    PROC main()
        Path_Draw;
    ENDPROC
    LOCAL PROC Path_Draw()
        MoveL point_0_clearance,v1000,fine,MyTool\WObj:=Workobject_1;
        MoveL point_0_contact,v1000,fine,MyTool\WObj:=Workobject_1;
        MoveL point_1_contact,v1000,fine,MyTool\WObj:=Workobject_1;
        MoveL point_1_clearance,v1000,fine,MyTool\WObj:=Workobject_1;
        MoveL point_2_clearance,v1000,fine,MyTool\WObj:=Workobject_1;
        MoveL point_2_contact,v1000,fine,MyTool\WObj:=Workobject_1;
        MoveL point_3_contact,v1000,fine,MyTool\WObj:=Workobject_1;
        MoveL point_3_clearance,v1000,fine,MyTool\WObj:=Workobject_1;
        MoveL point_4_clearance,v1000,fine,MyTool\WObj:=Workobject_1;
        MoveL point_4_contact,v1000,fine,MyTool\WObj:=Workobject_1;
        MoveL point_5_contact,v1000,fine,MyTool\WObj:=Workobject_1;
        MoveL point_5_clearance,v1000,fine,MyTool\WObj:=Workobject_1;
        MoveL point_6_clearance,v1000,fine,MyTool\WObj:=Workobject_1;
        MoveL point_6_contact,v1000,fine,MyTool\WObj:=Workobject_1;
        MoveL point_7_contact,v1000,fine,MyTool\WObj:=Workobject_1;
        MoveL point_7_clearance,v1000,fine,MyTool\WObj:=Workobject_1;
        MoveL point_8_clearance,v1000,fine,MyTool\WObj:=Workobject_1;
        MoveL point_8_contact,v1000,fine,MyTool\WObj:=Workobject_1;
        MoveL point_9_contact,v1000,fine,MyTool\WObj:=Workobject_1;
        MoveL point_9_clearance,v1000,fine,MyTool\WObj:=Workobject_1;
        MoveL point_10_clearance,v1000,fine,MyTool\WObj:=Workobject_1;
        MoveL point_10_contact,v1000,fine,MyTool\WObj:=Workobject_1;
        MoveL point_11_contact,v1000,fine,MyTool\WObj:=Workobject_1;
        MoveL point_11_clearance,v1000,fine,MyTool\WObj:=Workobject_1;
        MoveL point_12_clearance,v1000,fine,MyTool\WObj:=Workobject_1;
        MoveL point_12_contact,v1000,fine,MyTool\WObj:=Workobject_1;
        MoveL point_13_contact,v1000,fine,MyTool\WObj:=Workobject_1;
        MoveL point_13_clearance,v1000,fine,MyTool\WObj:=Workobject_1;
        MoveL point_14_clearance,v1000,fine,MyTool\WObj:=Workobject_1;
        MoveL point_14_contact,v1000,fine,MyTool\WObj:=Workobject_1;
        MoveL point_15_contact,v1000,fine,MyTool\WObj:=Workobject_1;
        MoveL point_15_clearance,v1000,fine,MyTool\WObj:=Workobject_1;
        MoveL point_16_clearance,v1000,fine,MyTool\WObj:=Workobject_1;
        MoveL point_16_contact,v1000,fine,MyTool\WObj:=Workobject_1;
        MoveL point_17_contact,v1000,fine,MyTool\WObj:=Workobject_1;
        MoveL point_17_clearance,v1000,fine,MyTool\WObj:=Workobject_1;
        MoveL point_18_clearance,v1000,fine,MyTool\WObj:=Workobject_1;
        MoveL point_18_contact,v1000,fine,MyTool\WObj:=Workobject_1;
        MoveL point_19_contact,v1000,fine,MyTool\WObj:=Workobject_1;
        MoveL point_19_clearance,v1000,fine,MyTool\WObj:=Workobject_1;
        MoveL point_20_clearance,v1000,fine,MyTool\WObj:=Workobject_1;
        MoveL point_20_contact,v1000,fine,MyTool\WObj:=Workobject_1;
        MoveL point_21_contact,v1000,fine,MyTool\WObj:=Workobject_1;
        MoveL point_21_clearance,v1000,fine,MyTool\WObj:=Workobject_1;
        MoveL point_22_clearance,v1000,fine,MyTool\WObj:=Workobject_1;
        MoveL point_22_contact,v1000,fine,MyTool\WObj:=Workobject_1;
        MoveL point_23_contact,v1000,fine,MyTool\WObj:=Workobject_1;
        MoveL point_23_clearance,v1000,fine,MyTool\WObj:=Workobject_1;
        MoveL point_24_clearance,v1000,fine,MyTool\WObj:=Workobject_1;
        MoveL point_24_contact,v1000,fine,MyTool\WObj:=Workobject_1;
        MoveL point_25_contact,v1000,fine,MyTool\WObj:=Workobject_1;
        MoveL point_25_clearance,v1000,fine,MyTool\WObj:=Workobject_1;
        MoveL point_26_clearance,v1000,fine,MyTool\WObj:=Workobject_1;
        MoveL point_26_contact,v1000,fine,MyTool\WObj:=Workobject_1;
        MoveL point_27_contact,v1000,fine,MyTool\WObj:=Workobject_1;
        MoveL point_27_clearance,v1000,fine,MyTool\WObj:=Workobject_1;
        MoveL point_28_clearance,v1000,fine,MyTool\WObj:=Workobject_1;
        MoveL point_28_contact,v1000,fine,MyTool\WObj:=Workobject_1;
        MoveL point_29_contact,v1000,fine,MyTool\WObj:=Workobject_1;
        MoveL point_29_clearance,v1000,fine,MyTool\WObj:=Workobject_1;
        MoveL point_30_clearance,v1000,fine,MyTool\WObj:=Workobject_1;
        MoveL point_30_contact,v1000,fine,MyTool\WObj:=Workobject_1;
        MoveL point_31_contact,v1000,fine,MyTool\WObj:=Workobject_1;
        MoveL point_31_clearance,v1000,fine,MyTool\WObj:=Workobject_1;
        MoveL point_32_clearance,v1000,fine,MyTool\WObj:=Workobject_1;
        MoveL point_32_contact,v1000,fine,MyTool\WObj:=Workobject_1;
        MoveL point_33_contact,v1000,fine,MyTool\WObj:=Workobject_1;
        MoveL point_33_clearance,v1000,fine,MyTool\WObj:=Workobject_1;
        MoveL point_34_clearance,v1000,fine,MyTool\WObj:=Workobject_1;
        MoveL point_34_contact,v1000,fine,MyTool\WObj:=Workobject_1;
        MoveL point_35_contact,v1000,fine,MyTool\WObj:=Workobject_1;
        MoveL point_35_clearance,v1000,fine,MyTool\WObj:=Workobject_1;
        MoveL point_36_clearance,v1000,fine,MyTool\WObj:=Workobject_1;
        MoveL point_36_contact,v1000,fine,MyTool\WObj:=Workobject_1;
        MoveL point_37_contact,v1000,fine,MyTool\WObj:=Workobject_1;
        MoveL point_37_clearance,v1000,fine,MyTool\WObj:=Workobject_1;
        MoveL point_38_clearance,v1000,fine,MyTool\WObj:=Workobject_1;
        MoveL point_38_contact,v1000,fine,MyTool\WObj:=Workobject_1;
        MoveL point_39_contact,v1000,fine,MyTool\WObj:=Workobject_1;
        MoveL point_39_clearance,v1000,fine,MyTool\WObj:=Workobject_1;
        MoveL point_40_clearance,v1000,fine,MyTool\WObj:=Workobject_1;
        MoveL point_40_contact,v1000,fine,MyTool\WObj:=Workobject_1;
        MoveL point_41_contact,v1000,fine,MyTool\WObj:=Workobject_1;
        MoveL point_41_clearance,v1000,fine,MyTool\WObj:=Workobject_1;
        MoveL point_42_clearance,v1000,fine,MyTool\WObj:=Workobject_1;
        MoveL point_42_contact,v1000,fine,MyTool\WObj:=Workobject_1;
        MoveL point_43_contact,v1000,fine,MyTool\WObj:=Workobject_1;
        MoveL point_43_clearance,v1000,fine,MyTool\WObj:=Workobject_1;
        MoveL point_44_clearance,v1000,fine,MyTool\WObj:=Workobject_1;
        MoveL point_44_contact,v1000,fine,MyTool\WObj:=Workobject_1;
        MoveL point_45_contact,v1000,fine,MyTool\WObj:=Workobject_1;
        MoveL point_45_clearance,v1000,fine,MyTool\WObj:=Workobject_1;
        MoveL point_46_clearance,v1000,fine,MyTool\WObj:=Workobject_1;
        MoveL point_46_contact,v1000,fine,MyTool\WObj:=Workobject_1;
        MoveL point_47_contact,v1000,fine,MyTool\WObj:=Workobject_1;
        MoveL point_47_clearance,v1000,fine,MyTool\WObj:=Workobject_1;
        MoveL point_48_clearance,v1000,fine,MyTool\WObj:=Workobject_1;
        MoveL point_48_contact,v1000,fine,MyTool\WObj:=Workobject_1;
        MoveL point_49_contact,v1000,fine,MyTool\WObj:=Workobject_1;
        MoveL point_49_clearance,v1000,fine,MyTool\WObj:=Workobject_1;
        MoveL point_50_clearance,v1000,fine,MyTool\WObj:=Workobject_1;
        MoveL point_50_contact,v1000,fine,MyTool\WObj:=Workobject_1;
        MoveL point_51_contact,v1000,fine,MyTool\WObj:=Workobject_1;
        MoveL point_51_clearance,v1000,fine,MyTool\WObj:=Workobject_1;
        MoveL point_52_clearance,v1000,fine,MyTool\WObj:=Workobject_1;
        MoveL point_52_contact,v1000,fine,MyTool\WObj:=Workobject_1;
        MoveL point_53_contact,v1000,fine,MyTool\WObj:=Workobject_1;
        MoveL point_53_clearance,v1000,fine,MyTool\WObj:=Workobject_1;
        MoveL point_54_clearance,v1000,fine,MyTool\WObj:=Workobject_1;
        MoveL point_54_contact,v1000,fine,MyTool\WObj:=Workobject_1;
        MoveL point_55_contact,v1000,fine,MyTool\WObj:=Workobject_1;
        MoveL point_55_clearance,v1000,fine,MyTool\WObj:=Workobject_1;
        MoveL point_56_clearance,v1000,fine,MyTool\WObj:=Workobject_1;
        MoveL point_56_contact,v1000,fine,MyTool\WObj:=Workobject_1;
        MoveL point_57_contact,v1000,fine,MyTool\WObj:=Workobject_1;
        MoveL point_57_clearance,v1000,fine,MyTool\WObj:=Workobject_1;
        MoveL point_58_clearance,v1000,fine,MyTool\WObj:=Workobject_1;
        MoveL point_58_contact,v1000,fine,MyTool\WObj:=Workobject_1;
        MoveL point_59_contact,v1000,fine,MyTool\WObj:=Workobject_1;
        MoveL point_59_clearance,v1000,fine,MyTool\WObj:=Workobject_1;
        MoveL point_60_clearance,v1000,fine,MyTool\WObj:=Workobject_1;
        MoveL point_60_contact,v1000,fine,MyTool\WObj:=Workobject_1;
        MoveL point_61_contact,v1000,fine,MyTool\WObj:=Workobject_1;
        MoveL point_61_clearance,v1000,fine,MyTool\WObj:=Workobject_1;
        MoveL point_62_clearance,v1000,fine,MyTool\WObj:=Workobject_1;
        MoveL point_62_contact,v1000,fine,MyTool\WObj:=Workobject_1;
        MoveL point_63_contact,v1000,fine,MyTool\WObj:=Workobject_1;
        MoveL point_63_clearance,v1000,fine,MyTool\WObj:=Workobject_1;
        MoveL point_64_clearance,v1000,fine,MyTool\WObj:=Workobject_1;
        MoveL point_64_contact,v1000,fine,MyTool\WObj:=Workobject_1;
        MoveL point_65_contact,v1000,fine,MyTool\WObj:=Workobject_1;
        MoveL point_65_clearance,v1000,fine,MyTool\WObj:=Workobject_1;
        MoveL point_66_clearance,v1000,fine,MyTool\WObj:=Workobject_1;
        MoveL point_66_contact,v1000,fine,MyTool\WObj:=Workobject_1;
        MoveL point_67_contact,v1000,fine,MyTool\WObj:=Workobject_1;
        MoveL point_67_clearance,v1000,fine,MyTool\WObj:=Workobject_1;
        MoveL point_68_clearance,v1000,fine,MyTool\WObj:=Workobject_1;
        MoveL point_68_contact,v1000,fine,MyTool\WObj:=Workobject_1;
        MoveL point_69_contact,v1000,fine,MyTool\WObj:=Workobject_1;
        MoveL point_69_clearance,v1000,fine,MyTool\WObj:=Workobject_1;
        MoveL point_70_clearance,v1000,fine,MyTool\WObj:=Workobject_1;
        MoveL point_70_contact,v1000,fine,MyTool\WObj:=Workobject_1;
        MoveL point_71_contact,v1000,fine,MyTool\WObj:=Workobject_1;
        MoveL point_71_clearance,v1000,fine,MyTool\WObj:=Workobject_1;
        MoveL point_72_clearance,v1000,fine,MyTool\WObj:=Workobject_1;
        MoveL point_72_contact,v1000,fine,MyTool\WObj:=Workobject_1;
        MoveL point_73_contact,v1000,fine,MyTool\WObj:=Workobject_1;
        MoveL point_73_clearance,v1000,fine,MyTool\WObj:=Workobject_1;
        MoveL point_74_clearance,v1000,fine,MyTool\WObj:=Workobject_1;
        MoveL point_74_contact,v1000,fine,MyTool\WObj:=Workobject_1;
        MoveL point_75_contact,v1000,fine,MyTool\WObj:=Workobject_1;
        MoveL point_75_clearance,v1000,fine,MyTool\WObj:=Workobject_1;
        MoveL point_76_clearance,v1000,fine,MyTool\WObj:=Workobject_1;
        MoveL point_76_contact,v1000,fine,MyTool\WObj:=Workobject_1;
        MoveL point_77_contact,v1000,fine,MyTool\WObj:=Workobject_1;
        MoveL point_77_clearance,v1000,fine,MyTool\WObj:=Workobject_1;
        MoveL point_78_clearance,v1000,fine,MyTool\WObj:=Workobject_1;
        MoveL point_78_contact,v1000,fine,MyTool\WObj:=Workobject_1;
        MoveL point_79_contact,v1000,fine,MyTool\WObj:=Workobject_1;
        MoveL point_79_clearance,v1000,fine,MyTool\WObj:=Workobject_1;
        MoveL point_80_clearance,v1000,fine,MyTool\WObj:=Workobject_1;
        MoveL point_80_contact,v1000,fine,MyTool\WObj:=Workobject_1;
        MoveL point_81_contact,v1000,fine,MyTool\WObj:=Workobject_1;
        MoveL point_81_clearance,v1000,fine,MyTool\WObj:=Workobject_1;
        MoveL point_82_clearance,v1000,fine,MyTool\WObj:=Workobject_1;
        MoveL point_82_contact,v1000,fine,MyTool\WObj:=Workobject_1;
        MoveL point_83_contact,v1000,fine,MyTool\WObj:=Workobject_1;
        MoveL point_83_clearance,v1000,fine,MyTool\WObj:=Workobject_1;
        MoveL point_84_clearance,v1000,fine,MyTool\WObj:=Workobject_1;
        MoveL point_84_contact,v1000,fine,MyTool\WObj:=Workobject_1;
        MoveL point_85_contact,v1000,fine,MyTool\WObj:=Workobject_1;
        MoveL point_85_clearance,v1000,fine,MyTool\WObj:=Workobject_1;
        MoveL point_86_clearance,v1000,fine,MyTool\WObj:=Workobject_1;
        MoveL point_86_contact,v1000,fine,MyTool\WObj:=Workobject_1;
        MoveL point_87_contact,v1000,fine,MyTool\WObj:=Workobject_1;
        MoveL point_87_clearance,v1000,fine,MyTool\WObj:=Workobject_1;
        MoveL point_88_clearance,v1000,fine,MyTool\WObj:=Workobject_1;
        MoveL point_88_contact,v1000,fine,MyTool\WObj:=Workobject_1;
        MoveL point_89_contact,v1000,fine,MyTool\WObj:=Workobject_1;
        MoveL point_89_clearance,v1000,fine,MyTool\WObj:=Workobject_1;
        MoveL point_90_clearance,v1000,fine,MyTool\WObj:=Workobject_1;
        MoveL point_90_contact,v1000,fine,MyTool\WObj:=Workobject_1;
        MoveL point_91_contact,v1000,fine,MyTool\WObj:=Workobject_1;
        MoveL point_91_clearance,v1000,fine,MyTool\WObj:=Workobject_1;
        MoveL point_92_clearance,v1000,fine,MyTool\WObj:=Workobject_1;
        MoveL point_92_contact,v1000,fine,MyTool\WObj:=Workobject_1;
        MoveL point_93_contact,v1000,fine,MyTool\WObj:=Workobject_1;
        MoveL point_93_clearance,v1000,fine,MyTool\WObj:=Workobject_1;
        MoveL point_94_clearance,v1000,fine,MyTool\WObj:=Workobject_1;
        MoveL point_94_contact,v1000,fine,MyTool\WObj:=Workobject_1;
        MoveL point_95_contact,v1000,fine,MyTool\WObj:=Workobject_1;
        MoveL point_95_clearance,v1000,fine,MyTool\WObj:=Workobject_1;
        MoveL point_96_clearance,v1000,fine,MyTool\WObj:=Workobject_1;
        MoveL point_96_contact,v1000,fine,MyTool\WObj:=Workobject_1;
        MoveL point_97_contact,v1000,fine,MyTool\WObj:=Workobject_1;
        MoveL point_97_clearance,v1000,fine,MyTool\WObj:=Workobject_1;
        MoveL point_98_clearance,v1000,fine,MyTool\WObj:=Workobject_1;
        MoveL point_98_contact,v1000,fine,MyTool\WObj:=Workobject_1;
        MoveL point_99_contact,v1000,fine,MyTool\WObj:=Workobject_1;
        MoveL point_99_clearance,v1000,fine,MyTool\WObj:=Workobject_1;
        MoveL point_100_clearance,v1000,fine,MyTool\WObj:=Workobject_1;
        MoveL point_100_contact,v1000,fine,MyTool\WObj:=Workobject_1;
        MoveL point_101_contact,v1000,fine,MyTool\WObj:=Workobject_1;
        MoveL point_101_clearance,v1000,fine,MyTool\WObj:=Workobject_1;
        MoveL point_102_clearance,v1000,fine,MyTool\WObj:=Workobject_1;
        MoveL point_102_contact,v1000,fine,MyTool\WObj:=Workobject_1;
        MoveL point_103_contact,v1000,fine,MyTool\WObj:=Workobject_1;
        MoveL point_103_clearance,v1000,fine,MyTool\WObj:=Workobject_1;
        MoveL point_104_clearance,v1000,fine,MyTool\WObj:=Workobject_1;
        MoveL point_104_contact,v1000,fine,MyTool\WObj:=Workobject_1;
        MoveL point_105_contact,v1000,fine,MyTool\WObj:=Workobject_1;
        MoveL point_105_clearance,v1000,fine,MyTool\WObj:=Workobject_1;
        MoveL point_106_clearance,v1000,fine,MyTool\WObj:=Workobject_1;
        MoveL point_106_contact,v1000,fine,MyTool\WObj:=Workobject_1;
        MoveL point_107_contact,v1000,fine,MyTool\WObj:=Workobject_1;
        MoveL point_107_clearance,v1000,fine,MyTool\WObj:=Workobject_1;
        MoveL point_108_clearance,v1000,fine,MyTool\WObj:=Workobject_1;
        MoveL point_108_contact,v1000,fine,MyTool\WObj:=Workobject_1;
        MoveL point_109_contact,v1000,fine,MyTool\WObj:=Workobject_1;
        MoveL point_109_clearance,v1000,fine,MyTool\WObj:=Workobject_1;
        MoveL point_110_clearance,v1000,fine,MyTool\WObj:=Workobject_1;
        MoveL point_110_contact,v1000,fine,MyTool\WObj:=Workobject_1;
        MoveL point_111_contact,v1000,fine,MyTool\WObj:=Workobject_1;
        MoveL point_111_clearance,v1000,fine,MyTool\WObj:=Workobject_1;
        MoveL point_112_clearance,v1000,fine,MyTool\WObj:=Workobject_1;
        MoveL point_112_contact,v1000,fine,MyTool\WObj:=Workobject_1;
        MoveL point_113_contact,v1000,fine,MyTool\WObj:=Workobject_1;
        MoveL point_113_clearance,v1000,fine,MyTool\WObj:=Workobject_1;
        MoveL point_114_clearance,v1000,fine,MyTool\WObj:=Workobject_1;
        MoveL point_114_contact,v1000,fine,MyTool\WObj:=Workobject_1;
        MoveL point_115_contact,v1000,fine,MyTool\WObj:=Workobject_1;
        MoveL point_115_clearance,v1000,fine,MyTool\WObj:=Workobject_1;
        MoveL point_116_clearance,v1000,fine,MyTool\WObj:=Workobject_1;
        MoveL point_116_contact,v1000,fine,MyTool\WObj:=Workobject_1;
        MoveL point_117_contact,v1000,fine,MyTool\WObj:=Workobject_1;
        MoveL point_117_clearance,v1000,fine,MyTool\WObj:=Workobject_1;
        MoveL point_118_clearance,v1000,fine,MyTool\WObj:=Workobject_1;
        MoveL point_118_contact,v1000,fine,MyTool\WObj:=Workobject_1;
        MoveL point_119_contact,v1000,fine,MyTool\WObj:=Workobject_1;
        MoveL point_119_clearance,v1000,fine,MyTool\WObj:=Workobject_1;
        MoveL point_120_clearance,v1000,fine,MyTool\WObj:=Workobject_1;
        MoveL point_120_contact,v1000,fine,MyTool\WObj:=Workobject_1;
        MoveL point_121_contact,v1000,fine,MyTool\WObj:=Workobject_1;
        MoveL point_121_clearance,v1000,fine,MyTool\WObj:=Workobject_1;
        MoveL point_122_clearance,v1000,fine,MyTool\WObj:=Workobject_1;
        MoveL point_122_contact,v1000,fine,MyTool\WObj:=Workobject_1;
        MoveL point_123_contact,v1000,fine,MyTool\WObj:=Workobject_1;
        MoveL point_123_clearance,v1000,fine,MyTool\WObj:=Workobject_1;
        MoveL point_124_clearance,v1000,fine,MyTool\WObj:=Workobject_1;
        MoveL point_124_contact,v1000,fine,MyTool\WObj:=Workobject_1;
        MoveL point_125_contact,v1000,fine,MyTool\WObj:=Workobject_1;
        MoveL point_125_clearance,v1000,fine,MyTool\WObj:=Workobject_1;
        MoveL point_126_clearance,v1000,fine,MyTool\WObj:=Workobject_1;
        MoveL point_126_contact,v1000,fine,MyTool\WObj:=Workobject_1;
        MoveL point_127_contact,v1000,fine,MyTool\WObj:=Workobject_1;
        MoveL point_127_clearance,v1000,fine,MyTool\WObj:=Workobject_1;
        MoveL point_128_clearance,v1000,fine,MyTool\WObj:=Workobject_1;
        MoveL point_128_contact,v1000,fine,MyTool\WObj:=Workobject_1;
        MoveL point_129_contact,v1000,fine,MyTool\WObj:=Workobject_1;
        MoveL point_129_clearance,v1000,fine,MyTool\WObj:=Workobject_1;
        MoveL point_130_clearance,v1000,fine,MyTool\WObj:=Workobject_1;
        MoveL point_130_contact,v1000,fine,MyTool\WObj:=Workobject_1;
        MoveL point_131_contact,v1000,fine,MyTool\WObj:=Workobject_1;
        MoveL point_131_clearance,v1000,fine,MyTool\WObj:=Workobject_1;
        MoveL point_132_clearance,v1000,fine,MyTool\WObj:=Workobject_1;
        MoveL point_132_contact,v1000,fine,MyTool\WObj:=Workobject_1;
        MoveL point_133_contact,v1000,fine,MyTool\WObj:=Workobject_1;
        MoveL point_133_clearance,v1000,fine,MyTool\WObj:=Workobject_1;
        MoveL point_134_clearance,v1000,fine,MyTool\WObj:=Workobject_1;
        MoveL point_134_contact,v1000,fine,MyTool\WObj:=Workobject_1;
        MoveL point_135_contact,v1000,fine,MyTool\WObj:=Workobject_1;
        MoveL point_135_clearance,v1000,fine,MyTool\WObj:=Workobject_1;
        MoveL point_136_clearance,v1000,fine,MyTool\WObj:=Workobject_1;
        MoveL point_136_contact,v1000,fine,MyTool\WObj:=Workobject_1;
        MoveL point_137_contact,v1000,fine,MyTool\WObj:=Workobject_1;
        MoveL point_137_clearance,v1000,fine,MyTool\WObj:=Workobject_1;
        MoveL point_138_clearance,v1000,fine,MyTool\WObj:=Workobject_1;
        MoveL point_138_contact,v1000,fine,MyTool\WObj:=Workobject_1;
        MoveL point_139_contact,v1000,fine,MyTool\WObj:=Workobject_1;
        MoveL point_139_clearance,v1000,fine,MyTool\WObj:=Workobject_1;
        MoveL point_140_clearance,v1000,fine,MyTool\WObj:=Workobject_1;
        MoveL point_140_contact,v1000,fine,MyTool\WObj:=Workobject_1;
        MoveL point_141_contact,v1000,fine,MyTool\WObj:=Workobject_1;
        MoveL point_141_clearance,v1000,fine,MyTool\WObj:=Workobject_1;
        MoveL point_142_clearance,v1000,fine,MyTool\WObj:=Workobject_1;
        MoveL point_142_contact,v1000,fine,MyTool\WObj:=Workobject_1;
        MoveL point_143_contact,v1000,fine,MyTool\WObj:=Workobject_1;
        MoveL point_143_clearance,v1000,fine,MyTool\WObj:=Workobject_1;
        MoveL point_144_clearance,v1000,fine,MyTool\WObj:=Workobject_1;
        MoveL point_144_contact,v1000,fine,MyTool\WObj:=Workobject_1;
        MoveL point_145_contact,v1000,fine,MyTool\WObj:=Workobject_1;
        MoveL point_145_clearance,v1000,fine,MyTool\WObj:=Workobject_1;
        MoveL point_146_clearance,v1000,fine,MyTool\WObj:=Workobject_1;
        MoveL point_146_contact,v1000,fine,MyTool\WObj:=Workobject_1;
        MoveL point_147_contact,v1000,fine,MyTool\WObj:=Workobject_1;
        MoveL point_147_clearance,v1000,fine,MyTool\WObj:=Workobject_1;
        MoveL point_148_clearance,v1000,fine,MyTool\WObj:=Workobject_1;
        MoveL point_148_contact,v1000,fine,MyTool\WObj:=Workobject_1;
        MoveL point_149_contact,v1000,fine,MyTool\WObj:=Workobject_1;
        MoveL point_149_clearance,v1000,fine,MyTool\WObj:=Workobject_1;
        MoveL point_150_clearance,v1000,fine,MyTool\WObj:=Workobject_1;
        MoveL point_150_contact,v1000,fine,MyTool\WObj:=Workobject_1;
        MoveL point_151_contact,v1000,fine,MyTool\WObj:=Workobject_1;
        MoveL point_151_clearance,v1000,fine,MyTool\WObj:=Workobject_1;
        MoveL point_152_clearance,v1000,fine,MyTool\WObj:=Workobject_1;
        MoveL point_152_contact,v1000,fine,MyTool\WObj:=Workobject_1;
        MoveL point_153_contact,v1000,fine,MyTool\WObj:=Workobject_1;
        MoveL point_153_clearance,v1000,fine,MyTool\WObj:=Workobject_1;
        MoveL point_154_clearance,v1000,fine,MyTool\WObj:=Workobject_1;
        MoveL point_154_contact,v1000,fine,MyTool\WObj:=Workobject_1;
        MoveL point_155_contact,v1000,fine,MyTool\WObj:=Workobject_1;
        MoveL point_155_clearance,v1000,fine,MyTool\WObj:=Workobject_1;
        MoveL point_156_clearance,v1000,fine,MyTool\WObj:=Workobject_1;
        MoveL point_156_contact,v1000,fine,MyTool\WObj:=Workobject_1;
        MoveL point_157_contact,v1000,fine,MyTool\WObj:=Workobject_1;
        MoveL point_157_clearance,v1000,fine,MyTool\WObj:=Workobject_1;
        MoveL point_158_clearance,v1000,fine,MyTool\WObj:=Workobject_1;
        MoveL point_158_contact,v1000,fine,MyTool\WObj:=Workobject_1;
        MoveL point_159_contact,v1000,fine,MyTool\WObj:=Workobject_1;
        MoveL point_159_clearance,v1000,fine,MyTool\WObj:=Workobject_1;
        MoveL point_160_clearance,v1000,fine,MyTool\WObj:=Workobject_1;
        MoveL point_160_contact,v1000,fine,MyTool\WObj:=Workobject_1;
        MoveL point_161_contact,v1000,fine,MyTool\WObj:=Workobject_1;
        MoveL point_161_clearance,v1000,fine,MyTool\WObj:=Workobject_1;
        MoveL point_162_clearance,v1000,fine,MyTool\WObj:=Workobject_1;
        MoveL point_162_contact,v1000,fine,MyTool\WObj:=Workobject_1;
        MoveL point_163_contact,v1000,fine,MyTool\WObj:=Workobject_1;
        MoveL point_163_clearance,v1000,fine,MyTool\WObj:=Workobject_1;
        MoveL point_164_clearance,v1000,fine,MyTool\WObj:=Workobject_1;
        MoveL point_164_contact,v1000,fine,MyTool\WObj:=Workobject_1;
        MoveL point_165_contact,v1000,fine,MyTool\WObj:=Workobject_1;
        MoveL point_165_clearance,v1000,fine,MyTool\WObj:=Workobject_1;
        MoveL point_166_clearance,v1000,fine,MyTool\WObj:=Workobject_1;
        MoveL point_166_contact,v1000,fine,MyTool\WObj:=Workobject_1;
        MoveL point_167_contact,v1000,fine,MyTool\WObj:=Workobject_1;
        MoveL point_167_clearance,v1000,fine,MyTool\WObj:=Workobject_1;
        MoveL point_168_clearance,v1000,fine,MyTool\WObj:=Workobject_1;
        MoveL point_168_contact,v1000,fine,MyTool\WObj:=Workobject_1;
        MoveL point_169_contact,v1000,fine,MyTool\WObj:=Workobject_1;
        MoveL point_169_clearance,v1000,fine,MyTool\WObj:=Workobject_1;
        MoveL point_170_clearance,v1000,fine,MyTool\WObj:=Workobject_1;
        MoveL point_170_contact,v1000,fine,MyTool\WObj:=Workobject_1;
        MoveL point_171_contact,v1000,fine,MyTool\WObj:=Workobject_1;
        MoveL point_171_clearance,v1000,fine,MyTool\WObj:=Workobject_1;
        MoveL point_172_clearance,v1000,fine,MyTool\WObj:=Workobject_1;
        MoveL point_172_contact,v1000,fine,MyTool\WObj:=Workobject_1;
        MoveL point_173_contact,v1000,fine,MyTool\WObj:=Workobject_1;
        MoveL point_173_clearance,v1000,fine,MyTool\WObj:=Workobject_1;
        MoveL point_174_clearance,v1000,fine,MyTool\WObj:=Workobject_1;
        MoveL point_174_contact,v1000,fine,MyTool\WObj:=Workobject_1;
        MoveL point_175_contact,v1000,fine,MyTool\WObj:=Workobject_1;
        MoveL point_175_clearance,v1000,fine,MyTool\WObj:=Workobject_1;
        MoveL point_176_clearance,v1000,fine,MyTool\WObj:=Workobject_1;
        MoveL point_176_contact,v1000,fine,MyTool\WObj:=Workobject_1;
        MoveL point_177_contact,v1000,fine,MyTool\WObj:=Workobject_1;
        MoveL point_177_clearance,v1000,fine,MyTool\WObj:=Workobject_1;
        MoveL point_178_clearance,v1000,fine,MyTool\WObj:=Workobject_1;
        MoveL point_178_contact,v1000,fine,MyTool\WObj:=Workobject_1;
        MoveL point_179_contact,v1000,fine,MyTool\WObj:=Workobject_1;
        MoveL point_179_clearance,v1000,fine,MyTool\WObj:=Workobject_1;
        MoveL point_180_clearance,v1000,fine,MyTool\WObj:=Workobject_1;
        MoveL point_180_contact,v1000,fine,MyTool\WObj:=Workobject_1;
        MoveL point_181_contact,v1000,fine,MyTool\WObj:=Workobject_1;
        MoveL point_181_clearance,v1000,fine,MyTool\WObj:=Workobject_1;
        MoveL point_182_clearance,v1000,fine,MyTool\WObj:=Workobject_1;
        MoveL point_182_contact,v1000,fine,MyTool\WObj:=Workobject_1;
        MoveL point_183_contact,v1000,fine,MyTool\WObj:=Workobject_1;
        MoveL point_183_clearance,v1000,fine,MyTool\WObj:=Workobject_1;
        MoveL point_184_clearance,v1000,fine,MyTool\WObj:=Workobject_1;
        MoveL point_184_contact,v1000,fine,MyTool\WObj:=Workobject_1;
        MoveL point_185_contact,v1000,fine,MyTool\WObj:=Workobject_1;
        MoveL point_185_clearance,v1000,fine,MyTool\WObj:=Workobject_1;
        MoveL point_186_clearance,v1000,fine,MyTool\WObj:=Workobject_1;
        MoveL point_186_contact,v1000,fine,MyTool\WObj:=Workobject_1;
        MoveL point_187_contact,v1000,fine,MyTool\WObj:=Workobject_1;
        MoveL point_187_clearance,v1000,fine,MyTool\WObj:=Workobject_1;
        MoveL point_188_clearance,v1000,fine,MyTool\WObj:=Workobject_1;
        MoveL point_188_contact,v1000,fine,MyTool\WObj:=Workobject_1;
        MoveL point_189_contact,v1000,fine,MyTool\WObj:=Workobject_1;
        MoveL point_189_clearance,v1000,fine,MyTool\WObj:=Workobject_1;
        MoveL point_190_clearance,v1000,fine,MyTool\WObj:=Workobject_1;
        MoveL point_190_contact,v1000,fine,MyTool\WObj:=Workobject_1;
        MoveL point_191_contact,v1000,fine,MyTool\WObj:=Workobject_1;
        MoveL point_191_clearance,v1000,fine,MyTool\WObj:=Workobject_1;
        MoveL point_192_clearance,v1000,fine,MyTool\WObj:=Workobject_1;
        MoveL point_192_contact,v1000,fine,MyTool\WObj:=Workobject_1;
        MoveL point_193_contact,v1000,fine,MyTool\WObj:=Workobject_1;
        MoveL point_193_clearance,v1000,fine,MyTool\WObj:=Workobject_1;
        MoveL point_194_clearance,v1000,fine,MyTool\WObj:=Workobject_1;
        MoveL point_194_contact,v1000,fine,MyTool\WObj:=Workobject_1;
        MoveL point_195_contact,v1000,fine,MyTool\WObj:=Workobject_1;
        MoveL point_195_clearance,v1000,fine,MyTool\WObj:=Workobject_1;
        MoveL point_196_clearance,v1000,fine,MyTool\WObj:=Workobject_1;
        MoveL point_196_contact,v1000,fine,MyTool\WObj:=Workobject_1;
        MoveL point_197_contact,v1000,fine,MyTool\WObj:=Workobject_1;
        MoveL point_197_clearance,v1000,fine,MyTool\WObj:=Workobject_1;
        MoveL point_198_clearance,v1000,fine,MyTool\WObj:=Workobject_1;
        MoveL point_198_contact,v1000,fine,MyTool\WObj:=Workobject_1;
        MoveL point_199_contact,v1000,fine,MyTool\WObj:=Workobject_1;
        MoveL point_199_clearance,v1000,fine,MyTool\WObj:=Workobject_1;
        MoveL point_200_clearance,v1000,fine,MyTool\WObj:=Workobject_1;
        MoveL point_200_contact,v1000,fine,MyTool\WObj:=Workobject_1;
        MoveL point_201_contact,v1000,fine,MyTool\WObj:=Workobject_1;
        MoveL point_201_clearance,v1000,fine,MyTool\WObj:=Workobject_1;
        MoveL point_202_clearance,v1000,fine,MyTool\WObj:=Workobject_1;
        MoveL point_202_contact,v1000,fine,MyTool\WObj:=Workobject_1;
        MoveL point_203_contact,v1000,fine,MyTool\WObj:=Workobject_1;
        MoveL point_203_clearance,v1000,fine,MyTool\WObj:=Workobject_1;
        MoveL point_204_clearance,v1000,fine,MyTool\WObj:=Workobject_1;
        MoveL point_204_contact,v1000,fine,MyTool\WObj:=Workobject_1;
        MoveL point_205_contact,v1000,fine,MyTool\WObj:=Workobject_1;
        MoveL point_205_clearance,v1000,fine,MyTool\WObj:=Workobject_1;
        MoveL point_206_clearance,v1000,fine,MyTool\WObj:=Workobject_1;
        MoveL point_206_contact,v1000,fine,MyTool\WObj:=Workobject_1;
        MoveL point_207_contact,v1000,fine,MyTool\WObj:=Workobject_1;
        MoveL point_207_clearance,v1000,fine,MyTool\WObj:=Workobject_1;
        MoveL point_208_clearance,v1000,fine,MyTool\WObj:=Workobject_1;
        MoveL point_208_contact,v1000,fine,MyTool\WObj:=Workobject_1;
        MoveL point_209_contact,v1000,fine,MyTool\WObj:=Workobject_1;
        MoveL point_209_clearance,v1000,fine,MyTool\WObj:=Workobject_1;
        MoveL point_210_clearance,v1000,fine,MyTool\WObj:=Workobject_1;
        MoveL point_210_contact,v1000,fine,MyTool\WObj:=Workobject_1;
        MoveL point_211_contact,v1000,fine,MyTool\WObj:=Workobject_1;
        MoveL point_211_clearance,v1000,fine,MyTool\WObj:=Workobject_1;
        MoveL point_212_clearance,v1000,fine,MyTool\WObj:=Workobject_1;
        MoveL point_212_contact,v1000,fine,MyTool\WObj:=Workobject_1;
        MoveL point_213_contact,v1000,fine,MyTool\WObj:=Workobject_1;
        MoveL point_213_clearance,v1000,fine,MyTool\WObj:=Workobject_1;
        MoveL point_214_clearance,v1000,fine,MyTool\WObj:=Workobject_1;
        MoveL point_214_contact,v1000,fine,MyTool\WObj:=Workobject_1;
        MoveL point_215_contact,v1000,fine,MyTool\WObj:=Workobject_1;
        MoveL point_215_clearance,v1000,fine,MyTool\WObj:=Workobject_1;
        MoveL point_216_clearance,v1000,fine,MyTool\WObj:=Workobject_1;
        MoveL point_216_contact,v1000,fine,MyTool\WObj:=Workobject_1;
        MoveL point_217_contact,v1000,fine,MyTool\WObj:=Workobject_1;
        MoveL point_217_clearance,v1000,fine,MyTool\WObj:=Workobject_1;
        MoveL point_218_clearance,v1000,fine,MyTool\WObj:=Workobject_1;
        MoveL point_218_contact,v1000,fine,MyTool\WObj:=Workobject_1;
        MoveL point_219_contact,v1000,fine,MyTool\WObj:=Workobject_1;
        MoveL point_219_clearance,v1000,fine,MyTool\WObj:=Workobject_1;
        MoveL point_220_clearance,v1000,fine,MyTool\WObj:=Workobject_1;
        MoveL point_220_contact,v1000,fine,MyTool\WObj:=Workobject_1;
        MoveL point_221_contact,v1000,fine,MyTool\WObj:=Workobject_1;
        MoveL point_221_clearance,v1000,fine,MyTool\WObj:=Workobject_1;
        MoveL point_222_clearance,v1000,fine,MyTool\WObj:=Workobject_1;
        MoveL point_222_contact,v1000,fine,MyTool\WObj:=Workobject_1;
        MoveL point_223_contact,v1000,fine,MyTool\WObj:=Workobject_1;
        MoveL point_223_clearance,v1000,fine,MyTool\WObj:=Workobject_1;
        MoveL point_224_clearance,v1000,fine,MyTool\WObj:=Workobject_1;
        MoveL point_224_contact,v1000,fine,MyTool\WObj:=Workobject_1;
        MoveL point_225_contact,v1000,fine,MyTool\WObj:=Workobject_1;
        MoveL point_225_clearance,v1000,fine,MyTool\WObj:=Workobject_1;
        MoveL point_226_clearance,v1000,fine,MyTool\WObj:=Workobject_1;
        MoveL point_226_contact,v1000,fine,MyTool\WObj:=Workobject_1;
        MoveL point_227_contact,v1000,fine,MyTool\WObj:=Workobject_1;
        MoveL point_227_clearance,v1000,fine,MyTool\WObj:=Workobject_1;
        MoveL point_228_clearance,v1000,fine,MyTool\WObj:=Workobject_1;
        MoveL point_228_contact,v1000,fine,MyTool\WObj:=Workobject_1;
        MoveL point_229_contact,v1000,fine,MyTool\WObj:=Workobject_1;
        MoveL point_229_clearance,v1000,fine,MyTool\WObj:=Workobject_1;
        MoveL point_230_clearance,v1000,fine,MyTool\WObj:=Workobject_1;
        MoveL point_230_contact,v1000,fine,MyTool\WObj:=Workobject_1;
        MoveL point_231_contact,v1000,fine,MyTool\WObj:=Workobject_1;
        MoveL point_231_clearance,v1000,fine,MyTool\WObj:=Workobject_1;
        MoveL point_232_clearance,v1000,fine,MyTool\WObj:=Workobject_1;
        MoveL point_232_contact,v1000,fine,MyTool\WObj:=Workobject_1;
        MoveL point_233_contact,v1000,fine,MyTool\WObj:=Workobject_1;
        MoveL point_233_clearance,v1000,fine,MyTool\WObj:=Workobject_1;
        MoveL point_234_clearance,v1000,fine,MyTool\WObj:=Workobject_1;
        MoveL point_234_contact,v1000,fine,MyTool\WObj:=Workobject_1;
        MoveL point_235_contact,v1000,fine,MyTool\WObj:=Workobject_1;
        MoveL point_235_clearance,v1000,fine,MyTool\WObj:=Workobject_1;
        MoveL point_236_clearance,v1000,fine,MyTool\WObj:=Workobject_1;
        MoveL point_236_contact,v1000,fine,MyTool\WObj:=Workobject_1;
        MoveL point_237_contact,v1000,fine,MyTool\WObj:=Workobject_1;
        MoveL point_237_clearance,v1000,fine,MyTool\WObj:=Workobject_1;
        MoveL point_238_clearance,v1000,fine,MyTool\WObj:=Workobject_1;
        MoveL point_238_contact,v1000,fine,MyTool\WObj:=Workobject_1;
        MoveL point_239_contact,v1000,fine,MyTool\WObj:=Workobject_1;
        MoveL point_239_clearance,v1000,fine,MyTool\WObj:=Workobject_1;
        MoveL point_240_clearance,v1000,fine,MyTool\WObj:=Workobject_1;
        MoveL point_240_contact,v1000,fine,MyTool\WObj:=Workobject_1;
        MoveL point_241_contact,v1000,fine,MyTool\WObj:=Workobject_1;
        MoveL point_241_clearance,v1000,fine,MyTool\WObj:=Workobject_1;
        MoveL point_242_clearance,v1000,fine,MyTool\WObj:=Workobject_1;
        MoveL point_242_contact,v1000,fine,MyTool\WObj:=Workobject_1;
        MoveL point_243_contact,v1000,fine,MyTool\WObj:=Workobject_1;
        MoveL point_243_clearance,v1000,fine,MyTool\WObj:=Workobject_1;
        MoveL point_244_clearance,v1000,fine,MyTool\WObj:=Workobject_1;
        MoveL point_244_contact,v1000,fine,MyTool\WObj:=Workobject_1;
        MoveL point_245_contact,v1000,fine,MyTool\WObj:=Workobject_1;
        MoveL point_245_clearance,v1000,fine,MyTool\WObj:=Workobject_1;
        MoveL point_246_clearance,v1000,fine,MyTool\WObj:=Workobject_1;
        MoveL point_246_contact,v1000,fine,MyTool\WObj:=Workobject_1;
        MoveL point_247_contact,v1000,fine,MyTool\WObj:=Workobject_1;
        MoveL point_247_clearance,v1000,fine,MyTool\WObj:=Workobject_1;
        MoveL point_248_clearance,v1000,fine,MyTool\WObj:=Workobject_1;
        MoveL point_248_contact,v1000,fine,MyTool\WObj:=Workobject_1;
        MoveL point_249_contact,v1000,fine,MyTool\WObj:=Workobject_1;
        MoveL point_249_clearance,v1000,fine,MyTool\WObj:=Workobject_1;
        MoveL point_250_clearance,v1000,fine,MyTool\WObj:=Workobject_1;
        MoveL point_250_contact,v1000,fine,MyTool\WObj:=Workobject_1;
        MoveL point_251_contact,v1000,fine,MyTool\WObj:=Workobject_1;
        MoveL point_251_clearance,v1000,fine,MyTool\WObj:=Workobject_1;
        MoveL point_252_clearance,v1000,fine,MyTool\WObj:=Workobject_1;
        MoveL point_252_contact,v1000,fine,MyTool\WObj:=Workobject_1;
        MoveL point_253_contact,v1000,fine,MyTool\WObj:=Workobject_1;
        MoveL point_253_clearance,v1000,fine,MyTool\WObj:=Workobject_1;
        MoveL point_254_clearance,v1000,fine,MyTool\WObj:=Workobject_1;
        MoveL point_254_contact,v1000,fine,MyTool\WObj:=Workobject_1;
        MoveL point_255_contact,v1000,fine,MyTool\WObj:=Workobject_1;
        MoveL point_255_clearance,v1000,fine,MyTool\WObj:=Workobject_1;
    ENDPROC
ENDMODULE

--- Backups/IRB_1600_8kg_1.45m/RAPID/TASK1/SYSMOD/LINKEDM.sys ---
%%%
  VERSION:1
  LANGUAGE:ENGLISH
%%%

MODULE LINKEDM (SYSMODULE)

! FOLLOWER
!     Name of electronically linked follower axis used by operator at teach pendent.
      PERS string l_f_axis_name{5}       :=  ["",  "", "", "", ""];

!     Name of the mechanical unit for follower axis.
      PERS string l_f_mecunt_n{5}  :=  ["", "", "", "", ""];

!     Linked follower axis number in the mechanical unit (first axis in mech. unit is number 1).
      PERS num l_f_axis_no{5}      :=  [0,          0,   0,  0,  0];

! MASTER
!     Name of the mechanical unit for linked master axis.
      PERS string l_m_mecunt_n{5} :=  ["", "", "", "", ""];

!     Linked master axis number in the mechanical unit (first axis in mech. unit is number 1).
!     See axis number table in documentation for different master mechanical units.
      PERS num l_m_axis_no{5}     :=  [0,  0,  0,  0,  0];

! POSITION OFFSET
!     The increase of the allowed offset position between the master and follower
!     positions, used when starting AUTO mode. As soon as the offset is decreased
!     the old configurated parameter is used.
!     Example: 3 => the configurated value of allowed offset is increased 3 times.
      PERS num offset_ratio{5}       :=  [10,  10,   10,  10,  10];

! SPEED RATIO
!     Speed_ratio used in AUTO and JOG modes [ very_slow   slow    normal    fast]
!     Value 1 = max allowed manual speed.
      CONST num speed_ratio {20}      := [0.01, 0.01, 0.01, 0.01, 0.01,
                                          0.05, 0.05, 0.05, 0.05, 0.05,
                                          0.20, 0.20, 0.20, 0.20, 0.20,
                                          1.00, 1.00, 1.00, 1.00, 1.00];

! STEP SIZE
!     Displacement position used in JOG mode for each activation of positive or
!     negative movement.                  [very_short    short   normal   long]
!     Unit degees or meter.
      CONST num displacement {20}     := [0.001, 0.001, 0.001, 0.001, 0.001,
                                          0.005, 0.005, 0.005, 0.005, 0.005,
                                          0.020, 0.020, 0.020, 0.020, 0.020,
                                          0.100, 0.100, 0.100, 0.100, 0.100];


!-------------------------------------------------------------
 PROC Linked_m ()
      Linked_m_exe ;
 ENDPROC
ENDMODULE
